TYPE (* ISOBUS UT Numeric Object (InputNumber/OutputNumber) pool properties *)
  (* Standard: 61499-2; Description: Copyright (c) 2026 Meisterschulen am Ostbahnhof This program and the accompanying materials are made available under the terms of the Eclipse Public License 2.0 which is available at https://www.eclipse.org/legal/epl-2.0/ SPDX-License-Identifier: EPL-2.0 *)
  (* Version 1.0, 2026-04-14, Franz Höpfinger, Meisterschulen am Ostbahnhof, initial API and implementation and/or initial documentation *)
  PACKAGE logiBUS::utils::conversion::phys;
  NumericObjectPool_S : STRUCT
    u16ObjId : UINT := 0; (* ISOBUS Object ID *)
    r32Scale : REAL := 1.0; (* Scale factor from object pool (e.g. 0.01) *)
    i32Offset : DINT := 0; (* Offset from object pool (e.g. -100000) *)
    u8Decimals : USINT := 0; (* Number of decimal places *)
  END_STRUCT;
END_TYPE
